(* Logix 5000 project; controller test vendor 1 type 14 code 196 rev 35.11; software revision 35.00 *)

TASK MainTask (continuous, watchdog 500 ms) : MainProgram

MODULES
   Local : vendor 1 type 14 code 196 (5069 0, rev 35.11)
END_MODULES

ADD_ON_INSTRUCTION Light_Temp_Hum_Control   (* revision 1.0 *)
VAR_INPUT
   Infrared_Sensor : BOOL; {required}
   Hum_Sensor : REAL; {required}
   Tem_Sensor : REAL; {required}
END_VAR
VAR_OUTPUT
   Light : BOOL; {access Read Only, visible}
   Dehumidifiers : BOOL; {visible}
   Air_Conditioner : BOOL; {visible}
END_VAR
VAR_INPUT
   Time_of_Day : DINT; {required}
END_VAR
VAR
   Time_Deactivation : TIMER := (PRE := 6000); {access None}
END_VAR

ROUTINE Logic   (* ladder *)
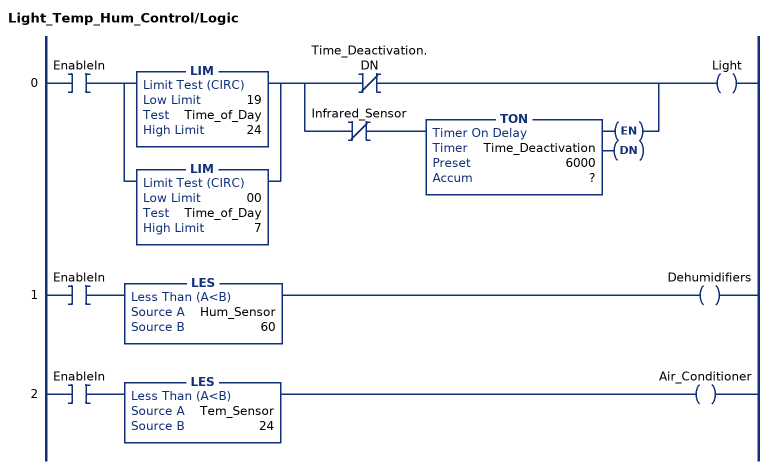
   0: XIC(EnableIn)[LIM(19,Time_of_Day,24) ,LIM(00,Time_of_Day,7) ][XIO(Time_Deactivation.DN) ,XIO(Infrared_Sensor) TON(Time_Deactivation,?,?) ]OTE(Light);
   1: XIC(EnableIn)LES(Hum_Sensor,60)OTE(Dehumidifiers);
   2: XIC(EnableIn)LES(Tem_Sensor,24)OTE(Air_Conditioner);
END_ROUTINE
END_ADD_ON_INSTRUCTION

PROGRAM MainProgram   (* main routine MainRoutine *)
VAR
   AI_Sen_Hum_1 : REAL;   // Humidity sensor area 1
   AI_Sen_Hum_2 : REAL;   // Humidity sensor area 2
   AI_Sen_Hum_3 : REAL;   // Humidity sensor area 3
   AI_Sen_Hum_4 : REAL;   // Humidity sensor area 4
   AI_Sen_Hum_5 : REAL;   // Humidity sensor area 5
   AI_Sen_Hum_6 : REAL;   // Humidity sensor area 6
   AI_Sen_Tem_1 : REAL;   // Temperature sensor area 1
   AI_Sen_Tem_2 : REAL;   // Temperature sensor area 2
   AI_Sen_Tem_3 : REAL;   // Temperature sensor area 3
   AI_Sen_Tem_4 : REAL;   // Temperature sensor area 4
   AI_Sen_Tem_5 : REAL;   // Temperature sensor area 5
   AI_Sen_Tem_6 : REAL := 1.0;   // Temperature sensor area 6
   Air_Conditioner_1 : BOOL;
   Air_Conditioner_2 : BOOL;
   Air_Conditioner_3 : BOOL;
   Air_Conditioner_4 : BOOL;
   Air_Conditioner_5 : BOOL;
   Air_Conditioner_6 : BOOL;
   Dehumidifiers_1 : BOOL;
   Dehumidifiers_2 : BOOL;
   Dehumidifiers_3 : BOOL;
   Dehumidifiers_4 : BOOL;
   Dehumidifiers_5 : BOOL;
   Dehumidifiers_6 : BOOL;
   Emergency_Stop : BOOL;
   I_Sen_IR_1 : BOOL;   // Infrared sensor area 1
   I_Sen_IR_2 : BOOL;   // Infrared sensor area 2
   I_Sen_IR_3 : BOOL;   // Infrared sensor area 3
   I_Sen_IR_4 : BOOL;   // Infrared sensor area 4
   I_Sen_IR_5 : BOOL;   // Infrared sensor area 5
   I_Sen_IR_6 : BOOL;   // Infrared sensor area 6
   I_Sen_IR_Parking : BOOL;   // Infrared sensor parking
   Key_Required : BOOL;
   LTHC_2 : Light_Temp_Hum_Control;
   LTHC_3 : Light_Temp_Hum_Control;
   LTHC_4 : Light_Temp_Hum_Control;
   LTHC_5 : Light_Temp_Hum_Control;
   LTHC_6 : Light_Temp_Hum_Control;
   O_Blinds : BOOL;   // Blinds
   O_Light_1 : BOOL;   // Light 1
   O_Light_2 : BOOL;   // Light 2
   O_Light_3 : BOOL;   // Light 3
   O_Light_4 : BOOL;   // Light 4
   O_Light_5 : BOOL;   // Light 5
   O_Light_6 : BOOL;   // Light 6
   O_Light_7 : BOOL;   // Gate
   Running : BOOL;
   Start_Button : BOOL;
   System_time : DINT[7];
        [5]   // Second
        [1]   // Month
        [2]   // Day
        [0]   // Year
        [3]   // Hour
        [4]   // Minute
        [6]   // MicroSecond
   Time_Deactivation : TIMER := (PRE := 6000);
END_VAR

ROUTINE MainRoutine   (* ladder *)
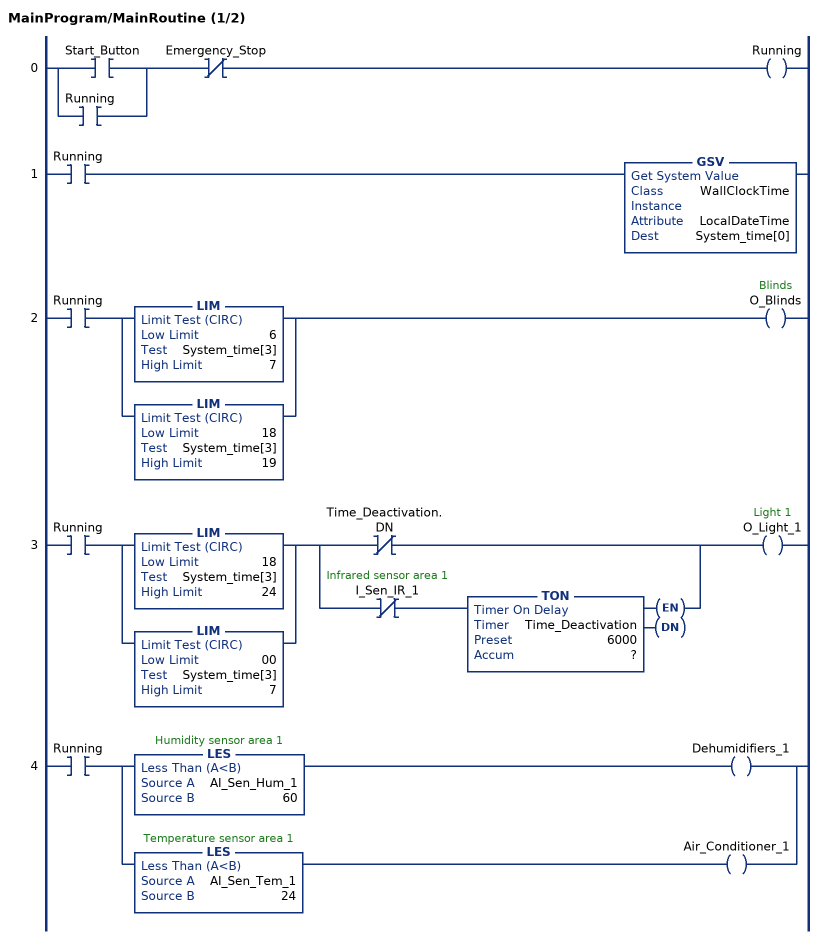
   0: [XIC(Start_Button) ,XIC(Running) ]XIO(Emergency_Stop)OTE(Running);
   1: XIC(Running)GSV(WallClockTime,,LocalDateTime,System_time[0]);
   2: XIC(Running)[LIM(6,System_time[3],7) ,LIM(18,System_time[3],19) ]OTE(O_Blinds);
   3: XIC(Running)[LIM(18,System_time[3],24) ,LIM(00,System_time[3],7) ][XIO(Time_Deactivation.DN) ,XIO(I_Sen_IR_1) TON(Time_Deactivation,?,?) ]OTE(O_Light_1);
   4: XIC(Running)[LES(AI_Sen_Hum_1,60) OTE(Dehumidifiers_1) ,LES(AI_Sen_Tem_1,24) OTE(Air_Conditioner_1) ];
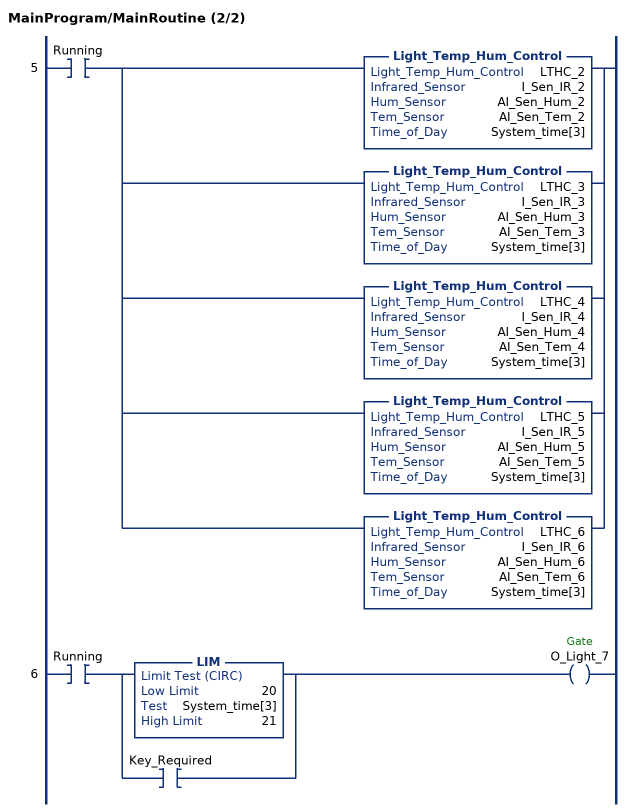
   5: XIC(Running)[Light_Temp_Hum_Control(LTHC_2,I_Sen_IR_2,AI_Sen_Hum_2,AI_Sen_Tem_2,System_time[3]) ,Light_Temp_Hum_Control(LTHC_3,I_Sen_IR_3,AI_Sen_Hum_3,AI_Sen_Tem_3,System_time[3]) ,Light_Temp_Hum_Control(LTHC_4,I_Sen_IR_4,AI_Sen_Hum_4,AI_Sen_Tem_4,System_time[3]) ,Light_Temp_Hum_Control(LTHC_5,I_Sen_IR_5,AI_Sen_Hum_5,AI_Sen_Tem_5,System_time[3]) ,Light_Temp_Hum_Control(LTHC_6,I_Sen_IR_6,AI_Sen_Hum_6,AI_Sen_Tem_6,System_time[3]) ];
   6: XIC(Running)[LIM(20,System_time[3],21) ,XIC(Key_Required) ]OTE(O_Light_7);
END_ROUTINE
END_PROGRAM
